FUNCTION_BLOCK ExtensionsCollection IMPLEMENTS I_ExtensionCollection
VAR
	extensions : Stack;
END_VAR

METHOD PUBLIC GetEnumerator : I_ForwardEnumerator
VAR_INPUT
END_VAR
GetEnumerator := extensions.GetEnumerator();
END_METHOD

METHOD PUBLIC Insert
VAR_INPUT
	ExtensionToAdd : I_Extension;
END_VAR
extensions.Push(ExtensionToAdd);
END_METHOD

METHOD PUBLIC TryGetByName : BOOL
VAR_INPUT
	Name : STRING;
	Destination : REFERENCE TO I_Extension;
END_VAR
VAR
	extensionEnumerator : I_ForwardEnumerator;
	currentExtension : I_Extension;
END_VAR
extensionEnumerator := extensions.GetEnumerator();

WHILE extensionEnumerator.MoveNext() DO 
	IF NOT extensionEnumerator.TryGet(currentExtension) THEN
		CONTINUE;
	END_IF
	
	IF currentExtension.Name = Name THEN 
		TryGetByName := TRUE;
		Destination := currentExtension;
		EXIT;
	END_IF

END_WHILE

extensionEnumerator.Dispose();
END_METHOD

END_FUNCTION_BLOCK

(* stored: Version 1.1.0.1, ProductVersion 3.1.4024.12
   POU ExtensionsCollection: Id {27384f57-a8c2-0737-00e0-7bb51765e0ee}, SpecialFunc None
   Method GetEnumerator: Id {2921e2e3-0729-0b2c-3db6-d5131b4b9730}
   Method Insert: Id {d4009a20-cf50-0b51-2df8-6eb5fce58568}
   Method TryGetByName: Id {02ffb6dc-d7f2-07ef-266b-097a2ed92420} *)
